PROGRAM MAIN
VAR
END_VAR

END_PROGRAM

(* stored: Version 1.1.0.1, ProductVersion 3.1.4024.12
   POU MAIN: Id {41bacaaa-6a51-06b5-3dc8-8773baf5c838}, SpecialFunc None *)
